Staubli VAL3: _WaitPartDyn.pgx

public program _WaitPartDyn()
// Wait part made in machine and mould fully open
begin
  //!brief
  // Wait for a part being made and conditions for the robot to enter mold.
  //
  call WaitPart(true)
end
